PROGRAM MAIN
VAR
	bToggle : BOOL;
END_VAR


bToggle := NOT bToggle;

END_PROGRAM

(* stored: Version 1.1.0.1, ProductVersion 3.1.4024.9
   POU MAIN: Id {3b0e438b-447a-4580-a659-8c765c101bdc}, SpecialFunc None *)
